PROGRAM MAIN
VAR	
	generateRecipe : BOOL;
	
	prepareData : PrepareData;
	addRecipeToDB : AddRecipeToDatabase;
	
	launch : Control;
END_VAR

IF generateRecipe THEN
	prepareData();
	//addRecipeToDB();
END_IF

END_PROGRAM

(* stored: Version 1.1.0.1, ProductVersion 3.1.4024.11
   POU MAIN: Id {bd7019dd-558f-4b28-a886-bdcf89182ad6}, SpecialFunc None *)
